INTERFACE itfReturnBOOL

METHOD mReturnBOOL : BOOL
VAR_INPUT
END_VAR
END_METHOD

END_INTERFACE

(* stored: Version 1.1.0.1, ProductVersion 3.1.4024.12
   Itf itfReturnBOOL: Id {513d6cf9-29a0-43a0-bab1-6f6a1dbb844a}
   Method mReturnBOOL: Id {81f6894f-c01b-46a3-a322-b598b865c488} *)
